{attribute 'GeneratedUsingTerminal: EL6002-0000-0019'}
{attribute addProperty BoxType "EL6002-0000-0019"}
{attribute addProperty Id "Transmit_requestBOOL1Receive_acceptedBOOL1Init_requestBOOL1Send_continuousBOOL1Output_lengthUSINT1"}
{attribute addProperty CRC "519785787"}
{attribute addProperty Size "5"}
TYPE Ctrl_1EFB4D3B :
STRUCT
	{attribute addProperty Name "Transmit_request"}
	Transmit_request : BOOL;
	{attribute addProperty Name "Receive_accepted"}
	Receive_accepted : BOOL;
	{attribute addProperty Name "Init_request"}
	Init_request : BOOL;
	{attribute addProperty Name "Send_continuous"}
	Send_continuous : BOOL;
	{attribute addProperty Name "Output_length"}
	Output_length : USINT;
END_STRUCT
END_TYPE

(* stored: Version 1.2.0.0, ProductVersion 3.1.4024.11
   DUT Ctrl_1EFB4D3B: Id {9f36bf55-0454-42ef-b1c4-46757c50863a} *)
